// Mitsubishi GX Developer project: PLC_PCO520L2   PLC: Q06UDEH

PROGRAM INPUT
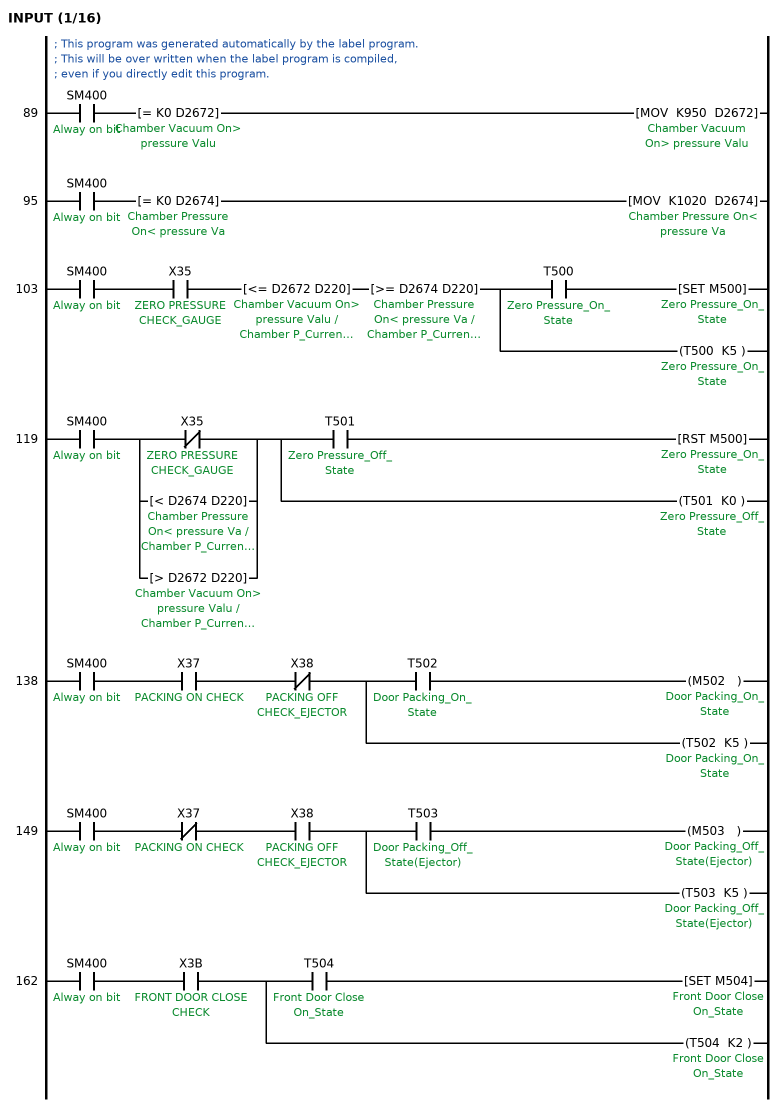
; This program was generated automatically by the label program.
; This will be over written when the label program is compiled,
; even if you directly edit this program.
89    LD      SM400  ; Alway on bit
      AND=    K0 D2672  ; Chamber Vacuum On> pressure Valu
      MOV     K950 D2672
95    LD      SM400  ; Alway on bit
      AND=    K0 D2674  ; Chamber Pressure On< pressure Va
      MOV     K1020 D2674
; 
103   LD      SM400  ; Alway on bit
      AND     X35  ; ZERO PRESSURE CHECK_GAUGE
      AND<=   D2672 D220  ; Chamber Vacuum On> pressure Valu / Chamber P_Current Pressure
      AND>=   D2674 D220  ; Chamber Pressure On< pressure Va / Chamber P_Current Pressure
      MPS
      AND     T500  ; Zero Pressure_On_State
      SET     M500  ; Zero Pressure_On_State
      MPP
      OUT     T500 K5  ; Zero Pressure_On_State
119   LD      SM400  ; Alway on bit
      LDI     X35  ; ZERO PRESSURE CHECK_GAUGE
      OR<     D2674 D220  ; Chamber Pressure On< pressure Va / Chamber P_Current Pressure
      OR>     D2672 D220  ; Chamber Vacuum On> pressure Valu / Chamber P_Current Pressure
      ANB
      MPS
      AND     T501  ; Zero Pressure_Off_State
      RST     M500  ; Zero Pressure_On_State
      MPP
      OUT     T501 K0  ; Zero Pressure_Off_State
; 
138   LD      SM400  ; Alway on bit
      AND     X37  ; PACKING ON CHECK
      ANI     X38  ; PACKING OFF CHECK_EJECTOR
      MPS
      AND     T502  ; Door Packing_On_State
      OUT     M502  ; Door Packing_On_State
      MPP
      OUT     T502 K5  ; Door Packing_On_State
149   LD      SM400  ; Alway on bit
      ANI     X37  ; PACKING ON CHECK
      AND     X38  ; PACKING OFF CHECK_EJECTOR
      MPS
      AND     T503  ; Door Packing_Off_State(Ejector)
      OUT     M503  ; Door Packing_Off_State(Ejector)
      MPP
      OUT     T503 K5  ; Door Packing_Off_State(Ejector)
; 
162   LD      SM400  ; Alway on bit
      AND     X3B  ; FRONT DOOR CLOSE CHECK
      MPS
      AND     T504  ; Front Door Close On_State
      SET     M504  ; Front Door Close On_State
      MPP
      OUT     T504 K2  ; Front Door Close On_State
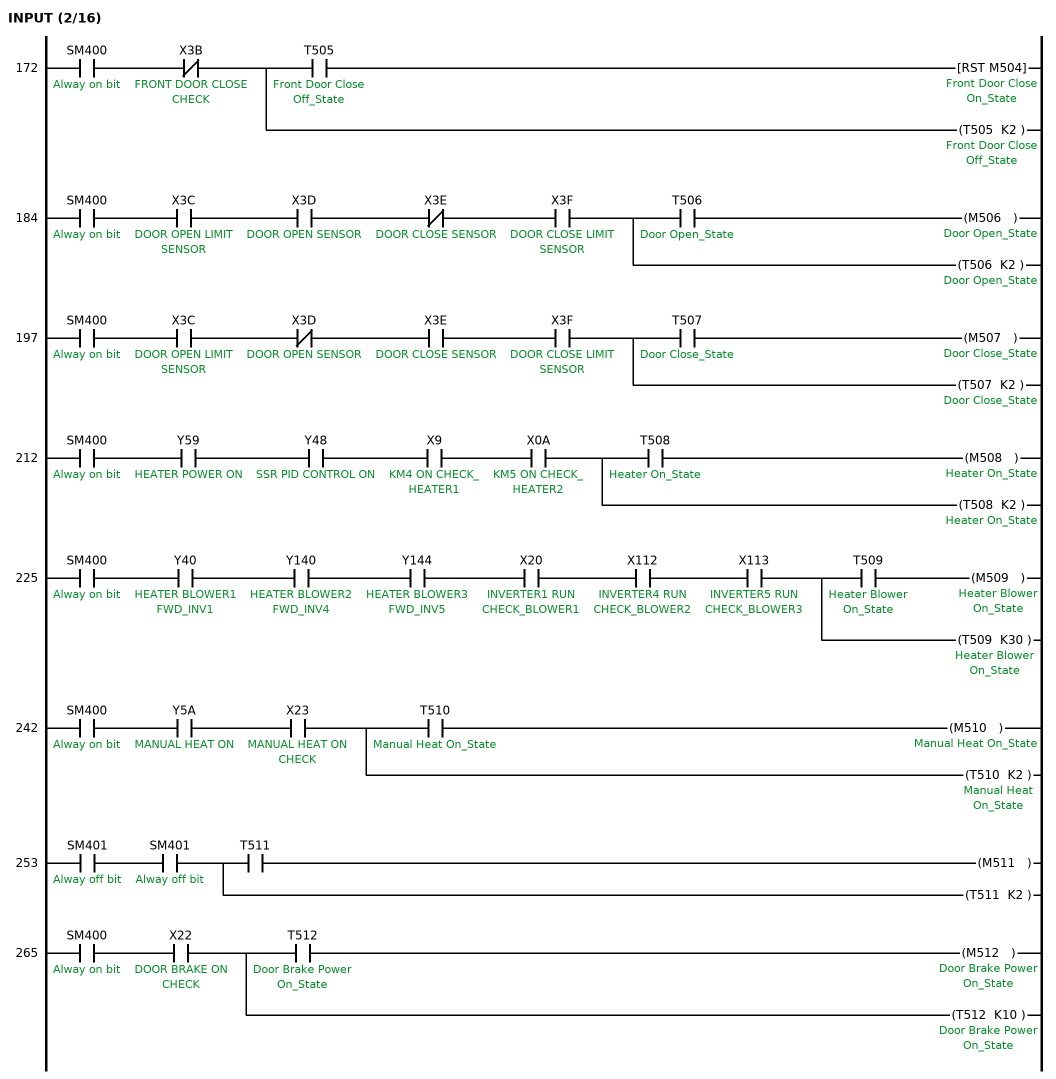
172   LD      SM400  ; Alway on bit
      ANI     X3B  ; FRONT DOOR CLOSE CHECK
      MPS
      AND     T505  ; Front Door Close Off_State
      RST     M504  ; Front Door Close On_State
      MPP
      OUT     T505 K2  ; Front Door Close Off_State
; 
184   LD      SM400  ; Alway on bit
      AND     X3C  ; DOOR OPEN LIMIT SENSOR
      AND     X3D  ; DOOR OPEN SENSOR
      ANI     X3E  ; DOOR CLOSE SENSOR
      AND     X3F  ; DOOR CLOSE LIMIT SENSOR
      MPS
      AND     T506  ; Door Open_State
      OUT     M506  ; Door Open_State
      MPP
      OUT     T506 K2  ; Door Open_State
197   LD      SM400  ; Alway on bit
      AND     X3C  ; DOOR OPEN LIMIT SENSOR
      ANI     X3D  ; DOOR OPEN SENSOR
      AND     X3E  ; DOOR CLOSE SENSOR
      AND     X3F  ; DOOR CLOSE LIMIT SENSOR
      MPS
      AND     T507  ; Door Close_State
      OUT     M507  ; Door Close_State
      MPP
      OUT     T507 K2  ; Door Close_State
; 
212   LD      SM400  ; Alway on bit
      AND     Y59  ; HEATER POWER ON
      AND     Y48  ; SSR PID CONTROL ON
      AND     X9  ; KM4 ON CHECK_HEATER1
      AND     X0A  ; KM5 ON CHECK_HEATER2
      MPS
      AND     T508  ; Heater On_State
      OUT     M508  ; Heater On_State
      MPP
      OUT     T508 K2  ; Heater On_State
225   LD      SM400  ; Alway on bit
      AND     Y40  ; HEATER BLOWER1 FWD_INV1
      AND     Y140  ; HEATER BLOWER2 FWD_INV4
      AND     Y144  ; HEATER BLOWER3 FWD_INV5
      AND     X20  ; INVERTER1 RUN CHECK_BLOWER1
      AND     X112  ; INVERTER4 RUN CHECK_BLOWER2
      AND     X113  ; INVERTER5 RUN CHECK_BLOWER3
      MPS
      AND     T509  ; Heater Blower On_State
      OUT     M509  ; Heater Blower On_State
      MPP
      OUT     T509 K30  ; Heater Blower On_State
; 
242   LD      SM400  ; Alway on bit
      AND     Y5A  ; MANUAL HEAT ON
      AND     X23  ; MANUAL HEAT ON CHECK
      MPS
      AND     T510  ; Manual Heat On_State
      OUT     M510  ; Manual Heat On_State
      MPP
      OUT     T510 K2  ; Manual Heat On_State
253   LD      SM401  ; Alway off bit
      AND     SM401  ; Alway off bit
      MPS
      AND     T511
      OUT     M511
      MPP
      OUT     T511 K2
; 
265   LD      SM400  ; Alway on bit
      AND     X22  ; DOOR BRAKE ON CHECK
      MPS
      AND     T512  ; Door Brake Power On_State
      OUT     M512  ; Door Brake Power On_State
      MPP
      OUT     T512 K10  ; Door Brake Power On_State
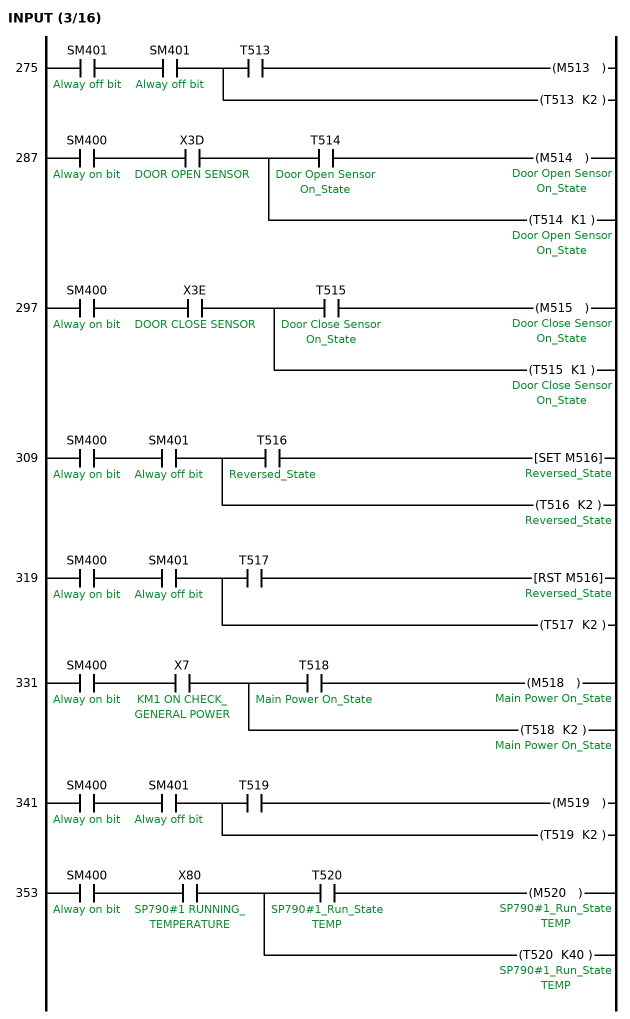
275   LD      SM401  ; Alway off bit
      AND     SM401  ; Alway off bit
      MPS
      AND     T513
      OUT     M513
      MPP
      OUT     T513 K2
; 
287   LD      SM400  ; Alway on bit
      AND     X3D  ; DOOR OPEN SENSOR
      MPS
      AND     T514  ; Door Open Sensor On_State
      OUT     M514  ; Door Open Sensor On_State
      MPP
      OUT     T514 K1  ; Door Open Sensor On_State
297   LD      SM400  ; Alway on bit
      AND     X3E  ; DOOR CLOSE SENSOR
      MPS
      AND     T515  ; Door Close Sensor On_State
      OUT     M515  ; Door Close Sensor On_State
      MPP
      OUT     T515 K1  ; Door Close Sensor On_State
; 
309   LD      SM400  ; Alway on bit
      AND     SM401  ; Alway off bit
      MPS
      AND     T516  ; Reversed_State
      SET     M516  ; Reversed_State
      MPP
      OUT     T516 K2  ; Reversed_State
319   LD      SM400  ; Alway on bit
      AND     SM401  ; Alway off bit
      MPS
      AND     T517
      RST     M516  ; Reversed_State
      MPP
      OUT     T517 K2
; 
331   LD      SM400  ; Alway on bit
      AND     X7  ; KM1 ON CHECK_GENERAL POWER
      MPS
      AND     T518  ; Main Power On_State
      OUT     M518  ; Main Power On_State
      MPP
      OUT     T518 K2  ; Main Power On_State
341   LD      SM400  ; Alway on bit
      AND     SM401  ; Alway off bit
      MPS
      AND     T519
      OUT     M519
      MPP
      OUT     T519 K2
; 
353   LD      SM400  ; Alway on bit
      AND     X80  ; SP790#1 RUNNING_TEMPERATURE
      MPS
      AND     T520  ; SP790#1_Run_State TEMP
      OUT     M520  ; SP790#1_Run_State TEMP
      MPP
      OUT     T520 K40  ; SP790#1_Run_State TEMP
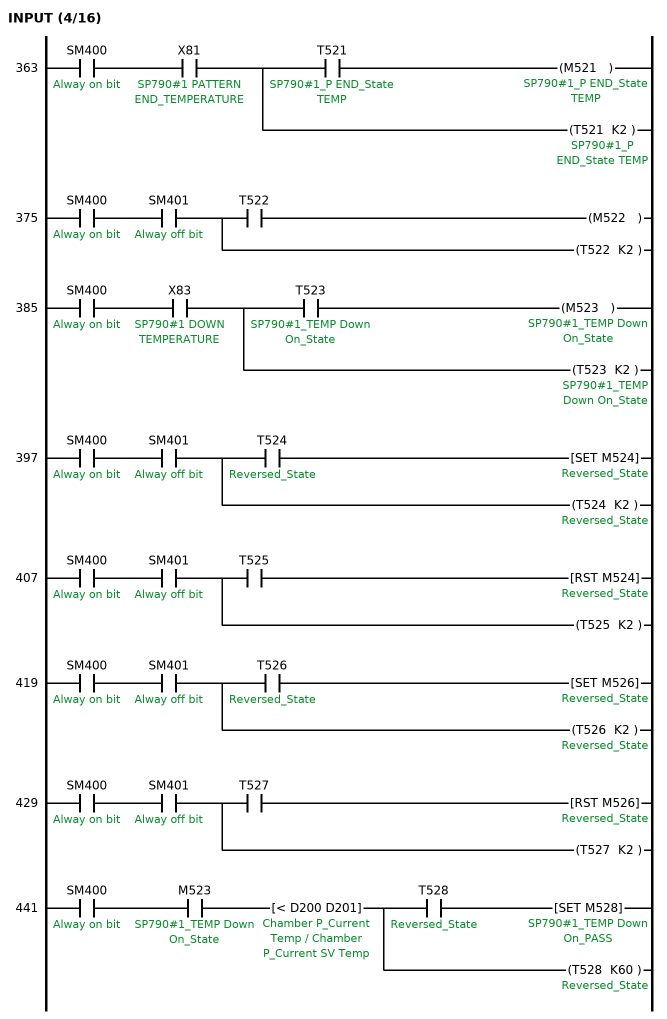
363   LD      SM400  ; Alway on bit
      AND     X81  ; SP790#1 PATTERN END_TEMPERATURE
      MPS
      AND     T521  ; SP790#1_P END_State TEMP
      OUT     M521  ; SP790#1_P END_State TEMP
      MPP
      OUT     T521 K2  ; SP790#1_P END_State TEMP
; 
375   LD      SM400  ; Alway on bit
      AND     SM401  ; Alway off bit
      MPS
      AND     T522
      OUT     M522
      MPP
      OUT     T522 K2
385   LD      SM400  ; Alway on bit
      AND     X83  ; SP790#1 DOWN TEMPERATURE
      MPS
      AND     T523  ; SP790#1_TEMP Down On_State
      OUT     M523  ; SP790#1_TEMP Down On_State
      MPP
      OUT     T523 K2  ; SP790#1_TEMP Down On_State
; 
397   LD      SM400  ; Alway on bit
      AND     SM401  ; Alway off bit
      MPS
      AND     T524  ; Reversed_State
      SET     M524  ; Reversed_State
      MPP
      OUT     T524 K2  ; Reversed_State
407   LD      SM400  ; Alway on bit
      AND     SM401  ; Alway off bit
      MPS
      AND     T525
      RST     M524  ; Reversed_State
      MPP
      OUT     T525 K2
; 
419   LD      SM400  ; Alway on bit
      AND     SM401  ; Alway off bit
      MPS
      AND     T526  ; Reversed_State
      SET     M526  ; Reversed_State
      MPP
      OUT     T526 K2  ; Reversed_State
429   LD      SM400  ; Alway on bit
      AND     SM401  ; Alway off bit
      MPS
      AND     T527
      RST     M526  ; Reversed_State
      MPP
      OUT     T527 K2
; 
441   LD      SM400  ; Alway on bit
      AND     M523  ; SP790#1_TEMP Down On_State
      AND<    D200 D201  ; Chamber P_Current Temp / Chamber P_Current SV Temp
      MPS
      AND     T528  ; Reversed_State
      SET     M528  ; SP790#1_TEMP Down On_PASS
      MPP
      OUT     T528 K60  ; Reversed_State
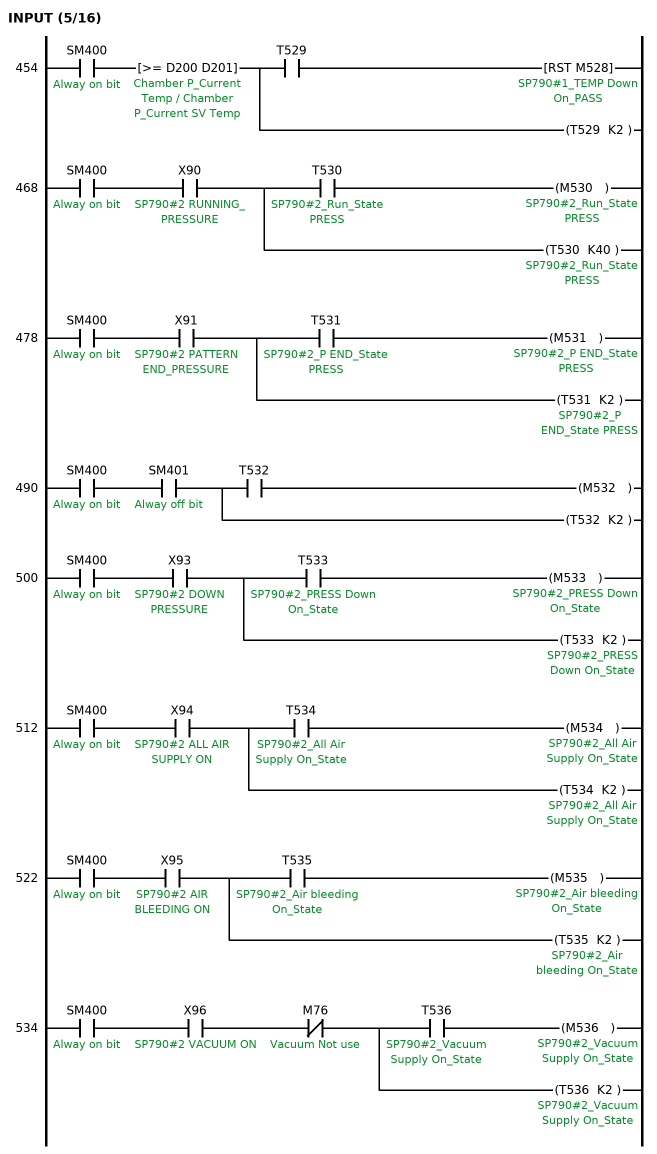
454   LD      SM400  ; Alway on bit
      AND>=   D200 D201  ; Chamber P_Current Temp / Chamber P_Current SV Temp
      MPS
      AND     T529
      RST     M528  ; SP790#1_TEMP Down On_PASS
      MPP
      OUT     T529 K2
; 
468   LD      SM400  ; Alway on bit
      AND     X90  ; SP790#2 RUNNING_PRESSURE
      MPS
      AND     T530  ; SP790#2_Run_State PRESS
      OUT     M530  ; SP790#2_Run_State PRESS
      MPP
      OUT     T530 K40  ; SP790#2_Run_State PRESS
478   LD      SM400  ; Alway on bit
      AND     X91  ; SP790#2 PATTERN END_PRESSURE
      MPS
      AND     T531  ; SP790#2_P END_State PRESS
      OUT     M531  ; SP790#2_P END_State PRESS
      MPP
      OUT     T531 K2  ; SP790#2_P END_State PRESS
; 
490   LD      SM400  ; Alway on bit
      AND     SM401  ; Alway off bit
      MPS
      AND     T532
      OUT     M532
      MPP
      OUT     T532 K2
500   LD      SM400  ; Alway on bit
      AND     X93  ; SP790#2 DOWN PRESSURE
      MPS
      AND     T533  ; SP790#2_PRESS Down On_State
      OUT     M533  ; SP790#2_PRESS Down On_State
      MPP
      OUT     T533 K2  ; SP790#2_PRESS Down On_State
; 
512   LD      SM400  ; Alway on bit
      AND     X94  ; SP790#2 ALL AIR SUPPLY ON
      MPS
      AND     T534  ; SP790#2_All Air Supply On_State
      OUT     M534  ; SP790#2_All Air Supply On_State
      MPP
      OUT     T534 K2  ; SP790#2_All Air Supply On_State
522   LD      SM400  ; Alway on bit
      AND     X95  ; SP790#2 AIR BLEEDING ON
      MPS
      AND     T535  ; SP790#2_Air bleeding On_State
      OUT     M535  ; SP790#2_Air bleeding On_State
      MPP
      OUT     T535 K2  ; SP790#2_Air bleeding On_State
; 
534   LD      SM400  ; Alway on bit
      AND     X96  ; SP790#2 VACUUM ON
      ANI     M76  ; Vacuum Not use
      MPS
      AND     T536  ; SP790#2_Vacuum Supply On_State
      OUT     M536  ; SP790#2_Vacuum Supply On_State
      MPP
      OUT     T536 K2  ; SP790#2_Vacuum Supply On_State
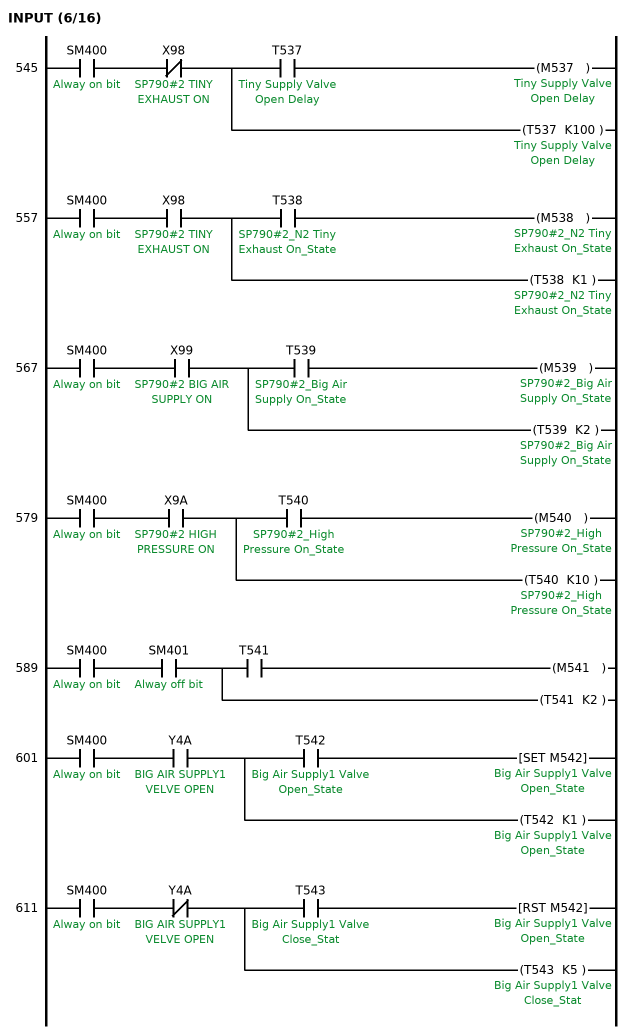
545   LD      SM400  ; Alway on bit
      ANI     X98  ; SP790#2 TINY EXHAUST ON
      MPS
      AND     T537  ; Tiny Supply Valve Open Delay
      OUT     M537  ; Tiny Supply Valve Open Delay
      MPP
      OUT     T537 K100  ; Tiny Supply Valve Open Delay
; 
557   LD      SM400  ; Alway on bit
      AND     X98  ; SP790#2 TINY EXHAUST ON
      MPS
      AND     T538  ; SP790#2_N2 Tiny Exhaust On_State
      OUT     M538  ; SP790#2_N2 Tiny Exhaust On_State
      MPP
      OUT     T538 K1  ; SP790#2_N2 Tiny Exhaust On_State
567   LD      SM400  ; Alway on bit
      AND     X99  ; SP790#2 BIG AIR SUPPLY ON
      MPS
      AND     T539  ; SP790#2_Big Air Supply On_State
      OUT     M539  ; SP790#2_Big Air Supply On_State
      MPP
      OUT     T539 K2  ; SP790#2_Big Air Supply On_State
; 
579   LD      SM400  ; Alway on bit
      AND     X9A  ; SP790#2 HIGH PRESSURE ON
      MPS
      AND     T540  ; SP790#2_High Pressure On_State
      OUT     M540  ; SP790#2_High Pressure On_State
      MPP
      OUT     T540 K10  ; SP790#2_High Pressure On_State
589   LD      SM400  ; Alway on bit
      AND     SM401  ; Alway off bit
      MPS
      AND     T541
      OUT     M541
      MPP
      OUT     T541 K2
; 
601   LD      SM400  ; Alway on bit
      AND     Y4A  ; BIG AIR SUPPLY1 VELVE OPEN
      MPS
      AND     T542  ; Big Air Supply1 Valve Open_State
      SET     M542  ; Big Air Supply1 Valve Open_State
      MPP
      OUT     T542 K1  ; Big Air Supply1 Valve Open_State
611   LD      SM400  ; Alway on bit
      ANI     Y4A  ; BIG AIR SUPPLY1 VELVE OPEN
      MPS
      AND     T543  ; Big Air Supply1 Valve Close_Stat
      RST     M542  ; Big Air Supply1 Valve Open_State
      MPP
      OUT     T543 K5  ; Big Air Supply1 Valve Close_Stat
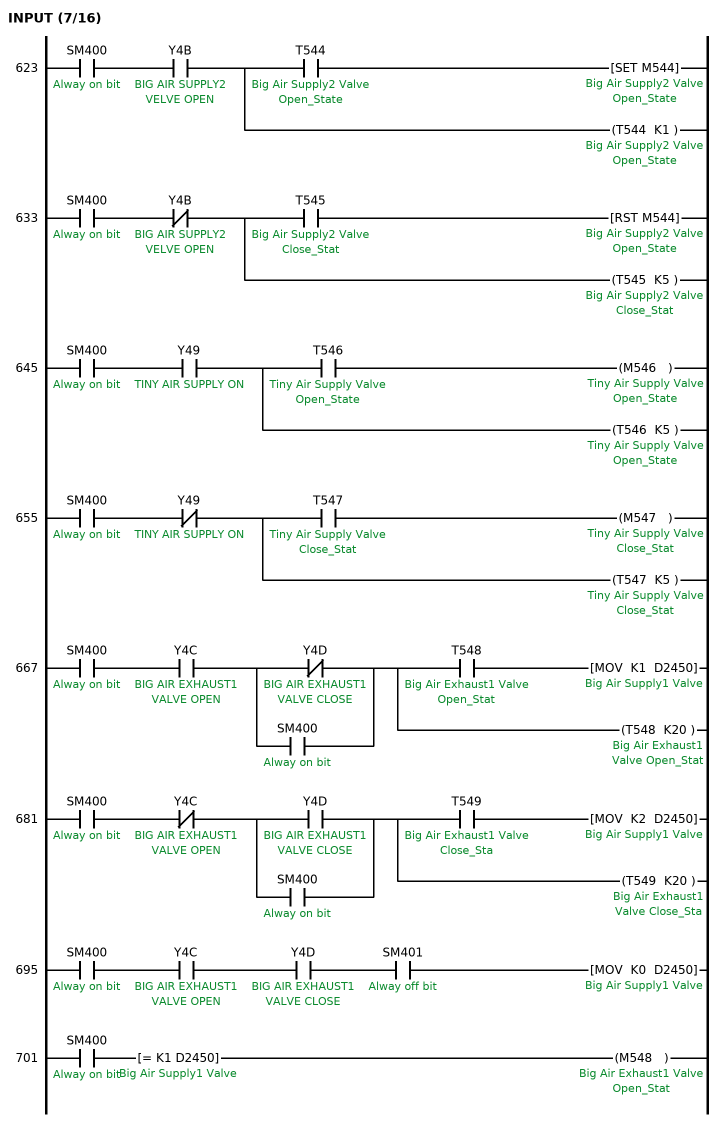
; 
623   LD      SM400  ; Alway on bit
      AND     Y4B  ; BIG AIR SUPPLY2 VELVE OPEN
      MPS
      AND     T544  ; Big Air Supply2 Valve Open_State
      SET     M544  ; Big Air Supply2 Valve Open_State
      MPP
      OUT     T544 K1  ; Big Air Supply2 Valve Open_State
633   LD      SM400  ; Alway on bit
      ANI     Y4B  ; BIG AIR SUPPLY2 VELVE OPEN
      MPS
      AND     T545  ; Big Air Supply2 Valve Close_Stat
      RST     M544  ; Big Air Supply2 Valve Open_State
      MPP
      OUT     T545 K5  ; Big Air Supply2 Valve Close_Stat
; 
645   LD      SM400  ; Alway on bit
      AND     Y49  ; TINY AIR SUPPLY ON
      MPS
      AND     T546  ; Tiny Air Supply Valve Open_State
      OUT     M546  ; Tiny Air Supply Valve Open_State
      MPP
      OUT     T546 K5  ; Tiny Air Supply Valve Open_State
655   LD      SM400  ; Alway on bit
      ANI     Y49  ; TINY AIR SUPPLY ON
      MPS
      AND     T547  ; Tiny Air Supply Valve Close_Stat
      OUT     M547  ; Tiny Air Supply Valve Close_Stat
      MPP
      OUT     T547 K5  ; Tiny Air Supply Valve Close_Stat
; 
667   LD      SM400  ; Alway on bit
      AND     Y4C  ; BIG AIR EXHAUST1 VALVE OPEN
      LDI     Y4D  ; BIG AIR EXHAUST1 VALVE CLOSE
      OR      SM400  ; Alway on bit
      ANB
      MPS
      AND     T548  ; Big Air Exhaust1 Valve Open_Stat
      MOV     K1 D2450  ; Big Air Supply1 Valve
      MPP
      OUT     T548 K20  ; Big Air Exhaust1 Valve Open_Stat
681   LD      SM400  ; Alway on bit
      ANI     Y4C  ; BIG AIR EXHAUST1 VALVE OPEN
      LD      Y4D  ; BIG AIR EXHAUST1 VALVE CLOSE
      OR      SM400  ; Alway on bit
      ANB
      MPS
      AND     T549  ; Big Air Exhaust1 Valve Close_Sta
      MOV     K2 D2450
      MPP
      OUT     T549 K20  ; Big Air Exhaust1 Valve Close_Sta
695   LD      SM400  ; Alway on bit
      AND     Y4C  ; BIG AIR EXHAUST1 VALVE OPEN
      AND     Y4D  ; BIG AIR EXHAUST1 VALVE CLOSE
      AND     SM401  ; Alway off bit
      MOV     K0 D2450
701   LD      SM400  ; Alway on bit
      AND=    K1 D2450  ; Big Air Supply1 Valve
      OUT     M548  ; Big Air Exhaust1 Valve Open_Stat
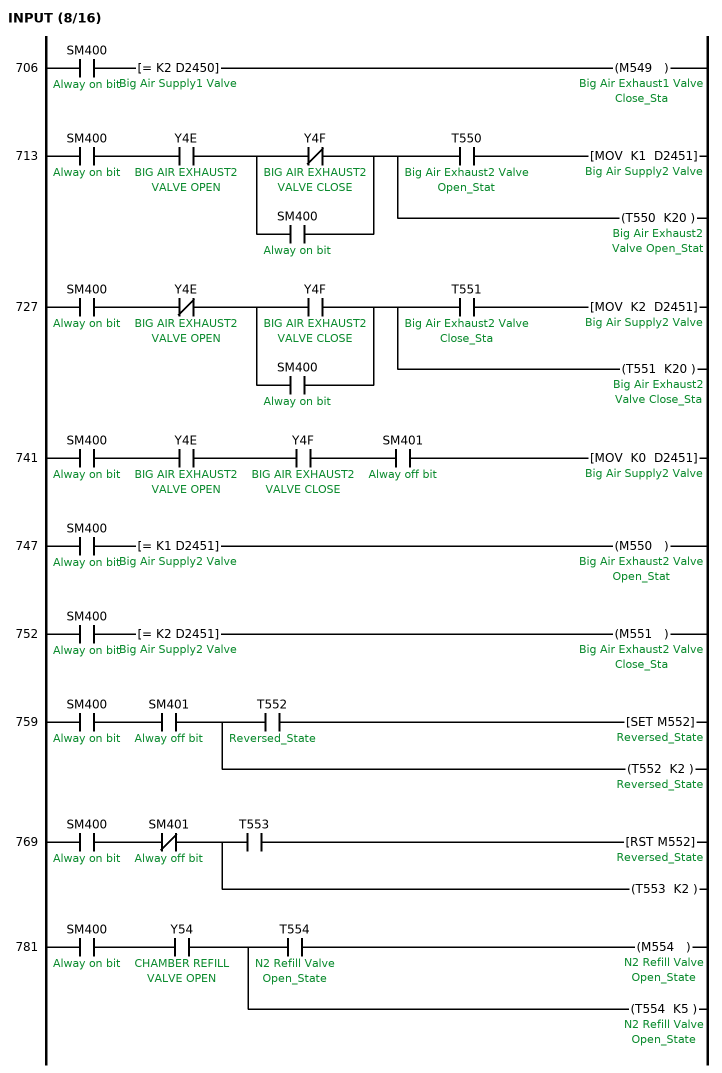
706   LD      SM400  ; Alway on bit
      AND=    K2 D2450  ; Big Air Supply1 Valve
      OUT     M549  ; Big Air Exhaust1 Valve Close_Sta
; 
713   LD      SM400  ; Alway on bit
      AND     Y4E  ; BIG AIR EXHAUST2 VALVE OPEN
      LDI     Y4F  ; BIG AIR EXHAUST2 VALVE CLOSE
      OR      SM400  ; Alway on bit
      ANB
      MPS
      AND     T550  ; Big Air Exhaust2 Valve Open_Stat
      MOV     K1 D2451  ; Big Air Supply2 Valve
      MPP
      OUT     T550 K20  ; Big Air Exhaust2 Valve Open_Stat
727   LD      SM400  ; Alway on bit
      ANI     Y4E  ; BIG AIR EXHAUST2 VALVE OPEN
      LD      Y4F  ; BIG AIR EXHAUST2 VALVE CLOSE
      OR      SM400  ; Alway on bit
      ANB
      MPS
      AND     T551  ; Big Air Exhaust2 Valve Close_Sta
      MOV     K2 D2451
      MPP
      OUT     T551 K20  ; Big Air Exhaust2 Valve Close_Sta
741   LD      SM400  ; Alway on bit
      AND     Y4E  ; BIG AIR EXHAUST2 VALVE OPEN
      AND     Y4F  ; BIG AIR EXHAUST2 VALVE CLOSE
      AND     SM401  ; Alway off bit
      MOV     K0 D2451
747   LD      SM400  ; Alway on bit
      AND=    K1 D2451  ; Big Air Supply2 Valve
      OUT     M550  ; Big Air Exhaust2 Valve Open_Stat
752   LD      SM400  ; Alway on bit
      AND=    K2 D2451  ; Big Air Supply2 Valve
      OUT     M551  ; Big Air Exhaust2 Valve Close_Sta
; 
759   LD      SM400  ; Alway on bit
      AND     SM401  ; Alway off bit
      MPS
      AND     T552  ; Reversed_State
      SET     M552  ; Reversed_State
      MPP
      OUT     T552 K2  ; Reversed_State
769   LD      SM400  ; Alway on bit
      ANI     SM401  ; Alway off bit
      MPS
      AND     T553
      RST     M552  ; Reversed_State
      MPP
      OUT     T553 K2
; 
781   LD      SM400  ; Alway on bit
      AND     Y54  ; CHAMBER REFILL VALVE OPEN
      MPS
      AND     T554  ; N2 Refill Valve Open_State
      OUT     M554  ; N2 Refill Valve Open_State
      MPP
      OUT     T554 K5  ; N2 Refill Valve Open_State
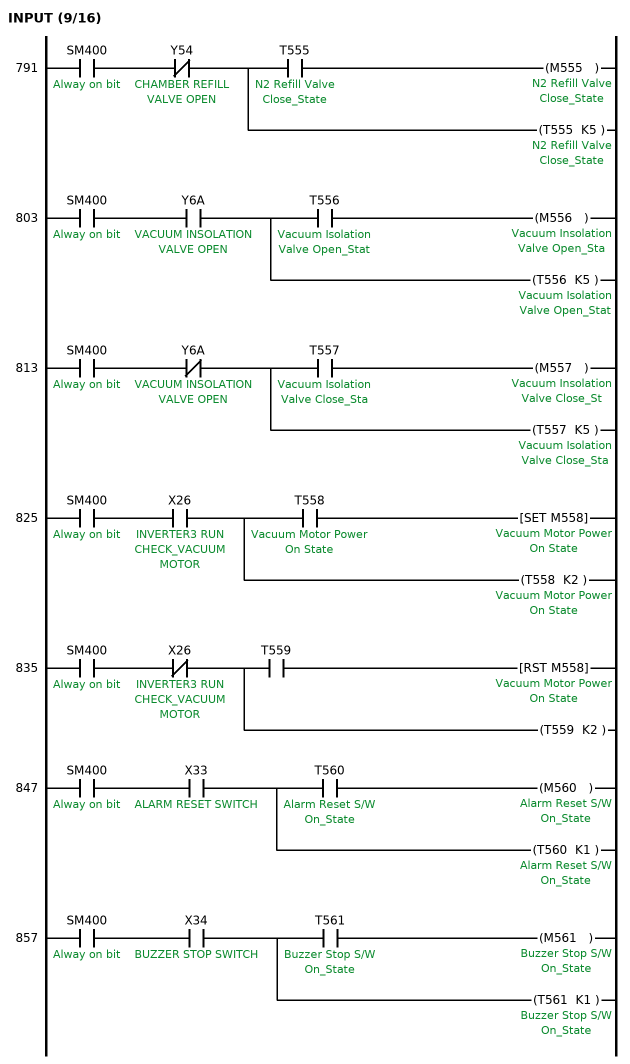
791   LD      SM400  ; Alway on bit
      ANI     Y54  ; CHAMBER REFILL VALVE OPEN
      MPS
      AND     T555  ; N2 Refill Valve Close_State
      OUT     M555  ; N2 Refill Valve Close_State
      MPP
      OUT     T555 K5  ; N2 Refill Valve Close_State
; 
803   LD      SM400  ; Alway on bit
      AND     Y6A  ; VACUUM INSOLATION VALVE OPEN
      MPS
      AND     T556  ; Vacuum Isolation Valve Open_Stat
      OUT     M556  ; Vacuum Insolation Valve Open_Sta
      MPP
      OUT     T556 K5  ; Vacuum Isolation Valve Open_Stat
813   LD      SM400  ; Alway on bit
      ANI     Y6A  ; VACUUM INSOLATION VALVE OPEN
      MPS
      AND     T557  ; Vacuum Isolation Valve Close_Sta
      OUT     M557  ; Vacuum Insolation Valve Close_St
      MPP
      OUT     T557 K5  ; Vacuum Isolation Valve Close_Sta
; 
825   LD      SM400  ; Alway on bit
      AND     X26  ; INVERTER3 RUN CHECK_VACUUM MOTOR
      MPS
      AND     T558  ; Vacuum Motor Power On State
      SET     M558  ; Vacuum Motor Power On State
      MPP
      OUT     T558 K2  ; Vacuum Motor Power On State
835   LD      SM400  ; Alway on bit
      ANI     X26  ; INVERTER3 RUN CHECK_VACUUM MOTOR
      MPS
      AND     T559
      RST     M558  ; Vacuum Motor Power On State
      MPP
      OUT     T559 K2
; 
847   LD      SM400  ; Alway on bit
      AND     X33  ; ALARM RESET SWITCH
      MPS
      AND     T560  ; Alarm Reset S/W On_State
      OUT     M560  ; Alarm Reset S/W On_State
      MPP
      OUT     T560 K1  ; Alarm Reset S/W On_State
857   LD      SM400  ; Alway on bit
      AND     X34  ; BUZZER STOP SWITCH
      MPS
      AND     T561  ; Buzzer Stop S/W On_State
      OUT     M561  ; Buzzer Stop S/W On_State
      MPP
      OUT     T561 K1  ; Buzzer Stop S/W On_State
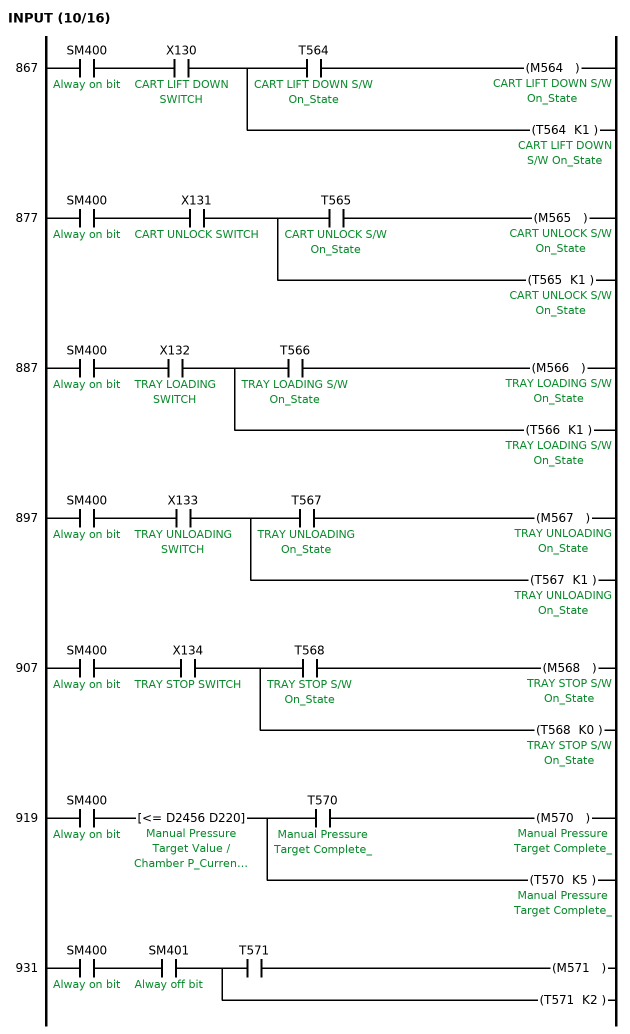
867   LD      SM400  ; Alway on bit
      AND     X130  ; CART LIFT DOWN SWITCH
      MPS
      AND     T564  ; CART LIFT DOWN S/W On_State
      OUT     M564  ; CART LIFT DOWN S/W On_State
      MPP
      OUT     T564 K1  ; CART LIFT DOWN S/W On_State
877   LD      SM400  ; Alway on bit
      AND     X131  ; CART UNLOCK SWITCH
      MPS
      AND     T565  ; CART UNLOCK S/W On_State
      OUT     M565  ; CART UNLOCK S/W On_State
      MPP
      OUT     T565 K1  ; CART UNLOCK S/W On_State
887   LD      SM400  ; Alway on bit
      AND     X132  ; TRAY LOADING SWITCH
      MPS
      AND     T566  ; TRAY LOADING S/W On_State
      OUT     M566  ; TRAY LOADING S/W On_State
      MPP
      OUT     T566 K1  ; TRAY LOADING S/W On_State
897   LD      SM400  ; Alway on bit
      AND     X133  ; TRAY UNLOADING SWITCH
      MPS
      AND     T567  ; TRAY UNLOADING On_State
      OUT     M567  ; TRAY UNLOADING On_State
      MPP
      OUT     T567 K1  ; TRAY UNLOADING On_State
907   LD      SM400  ; Alway on bit
      AND     X134  ; TRAY STOP SWITCH
      MPS
      AND     T568  ; TRAY STOP S/W On_State
      OUT     M568  ; TRAY STOP S/W On_State
      MPP
      OUT     T568 K0  ; TRAY STOP S/W On_State
; 
919   LD      SM400  ; Alway on bit
      AND<=   D2456 D220  ; Manual Pressure Target Value / Chamber P_Current Pressure
      MPS
      AND     T570  ; Manual Pressure Target Complete_
      OUT     M570  ; Manual Pressure Target Complete_
      MPP
      OUT     T570 K5  ; Manual Pressure Target Complete_
931   LD      SM400  ; Alway on bit
      AND     SM401  ; Alway off bit
      MPS
      AND     T571
      OUT     M571
      MPP
      OUT     T571 K2
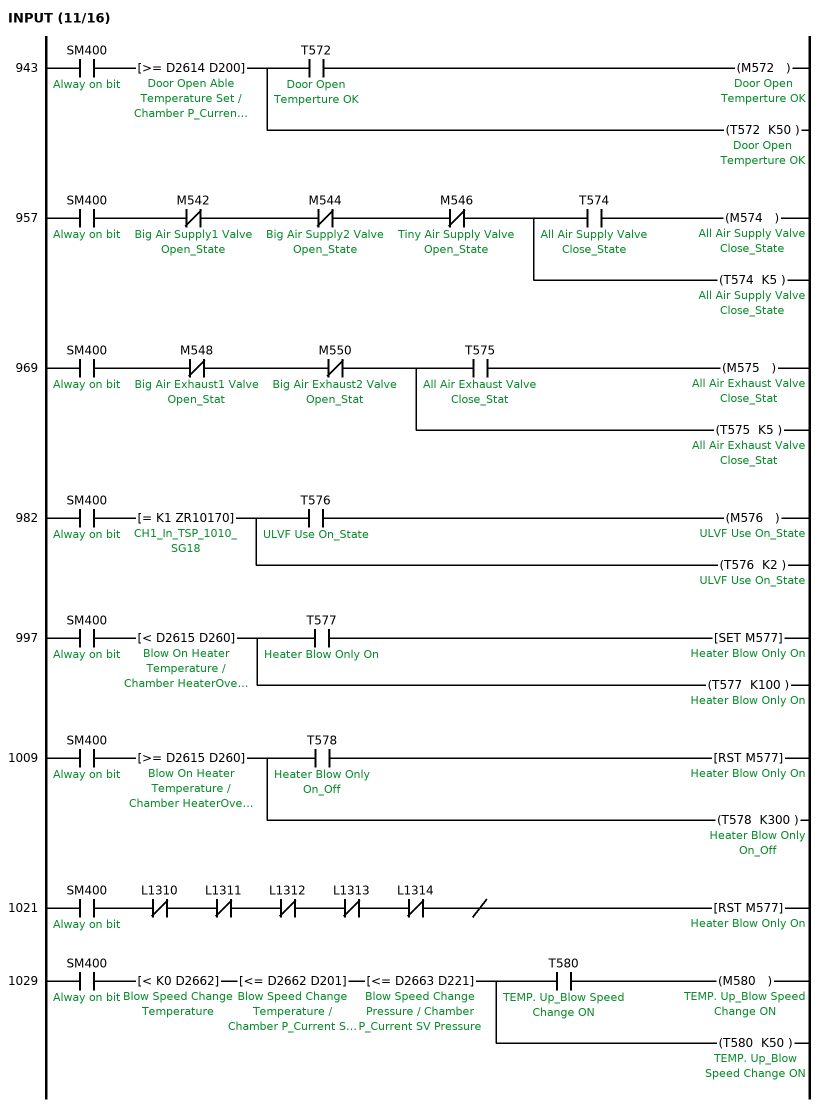
; 
943   LD      SM400  ; Alway on bit
      AND>=   D2614 D200  ; Door Open Able Temperature Set / Chamber P_Current Temp
      MPS
      AND     T572  ; Door Open Temperture OK
      OUT     M572  ; Door Open Temperture OK
      MPP
      OUT     T572 K50  ; Door Open Temperture OK
; 
957   LD      SM400  ; Alway on bit
      ANI     M542  ; Big Air Supply1 Valve Open_State
      ANI     M544  ; Big Air Supply2 Valve Open_State
      ANI     M546  ; Tiny Air Supply Valve Open_State
      MPS
      AND     T574  ; All Air Supply Valve Close_State
      OUT     M574  ; All Air Supply Valve Close_State
      MPP
      OUT     T574 K5  ; All Air Supply Valve Close_State
969   LD      SM400  ; Alway on bit
      ANI     M548  ; Big Air Exhaust1 Valve Open_Stat
      ANI     M550  ; Big Air Exhaust2 Valve Open_Stat
      MPS
      AND     T575  ; All Air Exhaust Valve Close_Stat
      OUT     M575  ; All Air Exhaust Valve Close_Stat
      MPP
      OUT     T575 K5  ; All Air Exhaust Valve Close_Stat
; 
982   LD      SM400  ; Alway on bit
      AND=    K1 ZR10170  ; CH1_In_TSP_1010_SG18
      MPS
      AND     T576  ; ULVF Use On_State
      OUT     M576  ; ULVF Use On_State
      MPP
      OUT     T576 K2  ; ULVF Use On_State
; 
997   LD      SM400  ; Alway on bit
      AND<    D2615 D260  ; Blow On Heater Temperature / Chamber HeaterOver Current Temp
      MPS
      AND     T577  ; Heater Blow Only On
      SET     M577  ; Heater Blow Only On
      MPP
      OUT     T577 K100  ; Heater Blow Only On
1009  LD      SM400  ; Alway on bit
      AND>=   D2615 D260  ; Blow On Heater Temperature / Chamber HeaterOver Current Temp
      MPS
      AND     T578  ; Heater Blow Only On_Off
      RST     M577  ; Heater Blow Only On
      MPP
      OUT     T578 K300  ; Heater Blow Only On_Off
1021  LD      SM400  ; Alway on bit
      ANI     L1310
      ANI     L1311
      ANI     L1312
      ANI     L1313
      ANI     L1314
      INV
      RST     M577  ; Heater Blow Only On
1029  LD      SM400  ; Alway on bit
      AND<    K0 D2662  ; Blow Speed Change Temperature
      AND<=   D2662 D201  ; Blow Speed Change Temperature / Chamber P_Current SV Temp
      AND<=   D2663 D221  ; Blow Speed Change Pressure / Chamber P_Current SV Pressure
      MPS
      AND     T580  ; TEMP. Up_Blow Speed Change ON
      OUT     M580  ; TEMP. Up_Blow Speed Change ON
      MPP
      OUT     T580 K50  ; TEMP. Up_Blow Speed Change ON
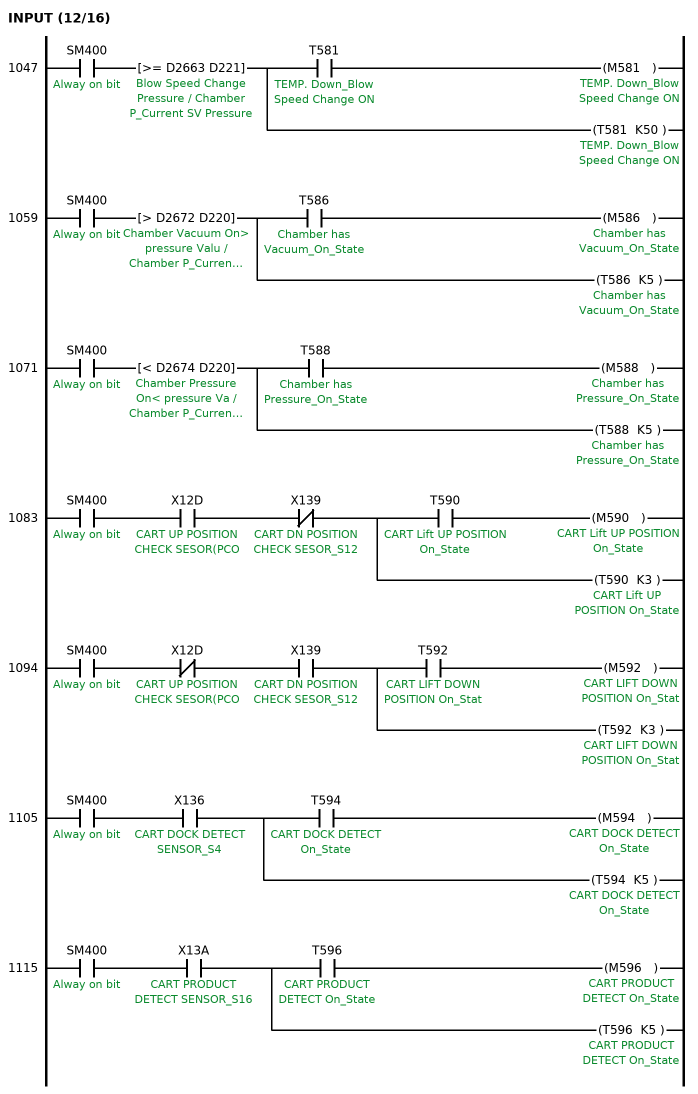
1047  LD      SM400  ; Alway on bit
      AND>=   D2663 D221  ; Blow Speed Change Pressure / Chamber P_Current SV Pressure
      MPS
      AND     T581  ; TEMP. Down_Blow Speed Change ON
      OUT     M581  ; TEMP. Down_Blow Speed Change ON
      MPP
      OUT     T581 K50  ; TEMP. Down_Blow Speed Change ON
1059  LD      SM400  ; Alway on bit
      AND>    D2672 D220  ; Chamber Vacuum On> pressure Valu / Chamber P_Current Pressure
      MPS
      AND     T586  ; Chamber has Vacuum_On_State
      OUT     M586  ; Chamber has Vacuum_On_State
      MPP
      OUT     T586 K5  ; Chamber has Vacuum_On_State
1071  LD      SM400  ; Alway on bit
      AND<    D2674 D220  ; Chamber Pressure On< pressure Va / Chamber P_Current Pressure
      MPS
      AND     T588  ; Chamber has Pressure_On_State
      OUT     M588  ; Chamber has Pressure_On_State
      MPP
      OUT     T588 K5  ; Chamber has Pressure_On_State
1083  LD      SM400  ; Alway on bit
      AND     X12D  ; CART UP POSITION CHECK SESOR(PCO
      ANI     X139  ; CART DN POSITION CHECK SESOR_S12
      MPS
      AND     T590  ; CART Lift UP POSITION On_State
      OUT     M590  ; CART Lift UP POSITION On_State
      MPP
      OUT     T590 K3  ; CART Lift UP POSITION On_State
1094  LD      SM400  ; Alway on bit
      ANI     X12D  ; CART UP POSITION CHECK SESOR(PCO
      AND     X139  ; CART DN POSITION CHECK SESOR_S12
      MPS
      AND     T592  ; CART LIFT DOWN  POSITION On_Stat
      OUT     M592  ; CART LIFT DOWN  POSITION On_Stat
      MPP
      OUT     T592 K3  ; CART LIFT DOWN  POSITION On_Stat
1105  LD      SM400  ; Alway on bit
      AND     X136  ; CART DOCK DETECT SENSOR_S4
      MPS
      AND     T594  ; CART DOCK DETECT On_State
      OUT     M594  ; CART DOCK DETECT On_State
      MPP
      OUT     T594 K5  ; CART DOCK DETECT On_State
1115  LD      SM400  ; Alway on bit
      AND     X13A  ; CART PRODUCT DETECT SENSOR_S16
      MPS
      AND     T596  ; CART PRODUCT DETECT On_State
      OUT     M596  ; CART PRODUCT DETECT On_State
      MPP
      OUT     T596 K5  ; CART PRODUCT DETECT On_State
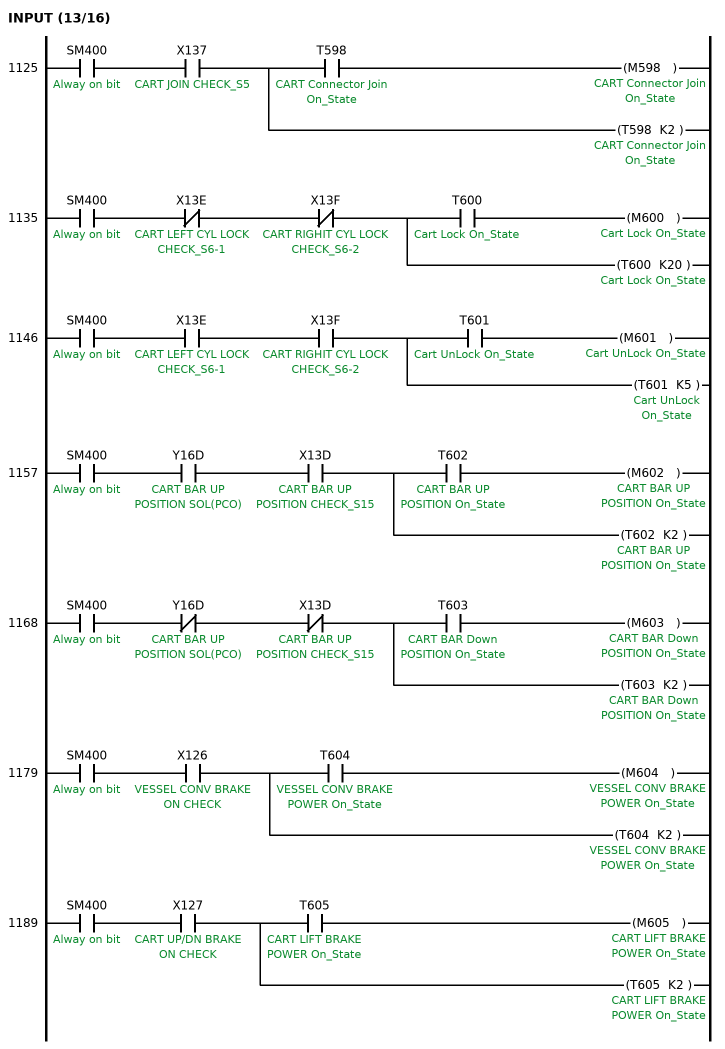
1125  LD      SM400  ; Alway on bit
      AND     X137  ; CART JOIN CHECK_S5
      MPS
      AND     T598  ; CART Connector Join On_State
      OUT     M598  ; CART Connector Join On_State
      MPP
      OUT     T598 K2  ; CART Connector Join On_State
1135  LD      SM400  ; Alway on bit
      ANI     X13E  ; CART LEFT CYL LOCK CHECK_S6-1
      ANI     X13F  ; CART RIGHIT CYL LOCK CHECK_S6-2
      MPS
      AND     T600  ; Cart Lock On_State
      OUT     M600  ; Cart Lock On_State
      MPP
      OUT     T600 K20  ; Cart Lock On_State
1146  LD      SM400  ; Alway on bit
      AND     X13E  ; CART LEFT CYL LOCK CHECK_S6-1
      AND     X13F  ; CART RIGHIT CYL LOCK CHECK_S6-2
      MPS
      AND     T601  ; Cart UnLock On_State
      OUT     M601  ; Cart UnLock On_State
      MPP
      OUT     T601 K5  ; Cart UnLock On_State
1157  LD      SM400  ; Alway on bit
      AND     Y16D  ; CART BAR UP POSITION SOL(PCO)
      AND     X13D  ; CART BAR UP POSITION CHECK_S15
      MPS
      AND     T602  ; CART BAR UP POSITION On_State
      OUT     M602  ; CART BAR UP POSITION On_State
      MPP
      OUT     T602 K2  ; CART BAR UP POSITION On_State
1168  LD      SM400  ; Alway on bit
      ANI     Y16D  ; CART BAR UP POSITION SOL(PCO)
      ANI     X13D  ; CART BAR UP POSITION CHECK_S15
      MPS
      AND     T603  ; CART BAR Down POSITION On_State
      OUT     M603  ; CART BAR Down POSITION On_State
      MPP
      OUT     T603 K2  ; CART BAR Down POSITION On_State
1179  LD      SM400  ; Alway on bit
      AND     X126  ; VESSEL CONV BRAKE ON CHECK
      MPS
      AND     T604  ; VESSEL CONV BRAKE POWER On_State
      OUT     M604  ; VESSEL CONV BRAKE POWER On_State
      MPP
      OUT     T604 K2  ; VESSEL CONV BRAKE POWER On_State
1189  LD      SM400  ; Alway on bit
      AND     X127  ; CART UP/DN BRAKE ON CHECK
      MPS
      AND     T605  ; CART LIFT BRAKE POWER On_State
      OUT     M605  ; CART LIFT BRAKE POWER On_State
      MPP
      OUT     T605 K2  ; CART LIFT BRAKE POWER On_State
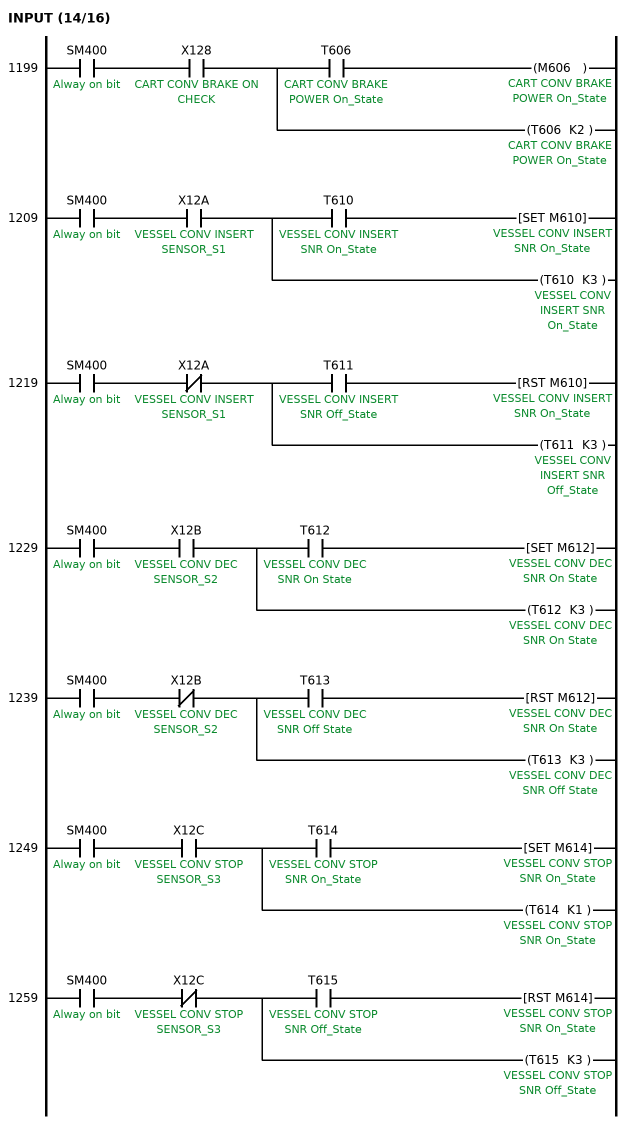
1199  LD      SM400  ; Alway on bit
      AND     X128  ; CART CONV BRAKE ON CHECK
      MPS
      AND     T606  ; CART CONV BRAKE POWER On_State
      OUT     M606  ; CART CONV BRAKE POWER On_State
      MPP
      OUT     T606 K2  ; CART CONV BRAKE POWER On_State
1209  LD      SM400  ; Alway on bit
      AND     X12A  ; VESSEL CONV INSERT SENSOR_S1
      MPS
      AND     T610  ; VESSEL CONV INSERT SNR On_State
      SET     M610  ; VESSEL CONV INSERT SNR On_State
      MPP
      OUT     T610 K3  ; VESSEL CONV INSERT SNR On_State
1219  LD      SM400  ; Alway on bit
      ANI     X12A  ; VESSEL CONV INSERT SENSOR_S1
      MPS
      AND     T611  ; VESSEL CONV INSERT SNR Off_State
      RST     M610  ; VESSEL CONV INSERT SNR On_State
      MPP
      OUT     T611 K3  ; VESSEL CONV INSERT SNR Off_State
1229  LD      SM400  ; Alway on bit
      AND     X12B  ; VESSEL CONV DEC SENSOR_S2
      MPS
      AND     T612  ; VESSEL CONV DEC SNR On State
      SET     M612  ; VESSEL CONV DEC SNR On State
      MPP
      OUT     T612 K3  ; VESSEL CONV DEC SNR On State
1239  LD      SM400  ; Alway on bit
      ANI     X12B  ; VESSEL CONV DEC SENSOR_S2
      MPS
      AND     T613  ; VESSEL CONV DEC SNR Off State
      RST     M612  ; VESSEL CONV DEC SNR On State
      MPP
      OUT     T613 K3  ; VESSEL CONV DEC SNR Off State
1249  LD      SM400  ; Alway on bit
      AND     X12C  ; VESSEL CONV STOP SENSOR_S3
      MPS
      AND     T614  ; VESSEL CONV STOP SNR On_State
      SET     M614  ; VESSEL CONV STOP SNR On_State
      MPP
      OUT     T614 K1  ; VESSEL CONV STOP SNR On_State
1259  LD      SM400  ; Alway on bit
      ANI     X12C  ; VESSEL CONV STOP SENSOR_S3
      MPS
      AND     T615  ; VESSEL CONV STOP SNR Off_State
      RST     M614  ; VESSEL CONV STOP SNR On_State
      MPP
      OUT     T615 K3  ; VESSEL CONV STOP SNR Off_State
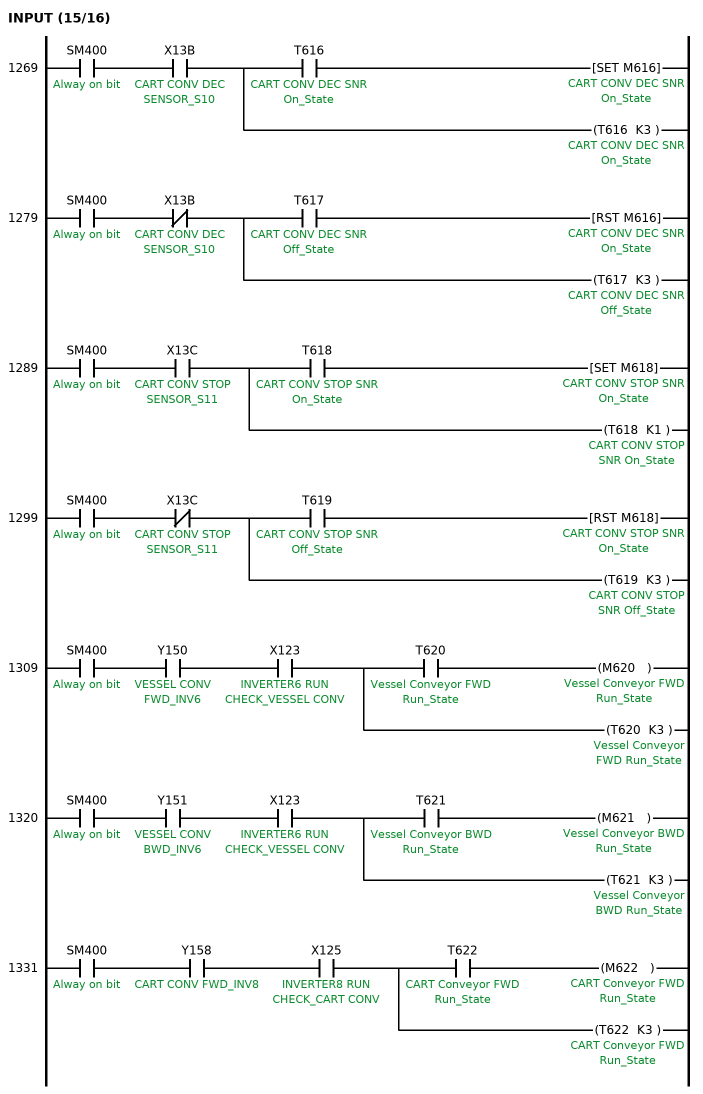
1269  LD      SM400  ; Alway on bit
      AND     X13B  ; CART CONV DEC SENSOR_S10
      MPS
      AND     T616  ; CART CONV DEC SNR On_State
      SET     M616  ; CART CONV DEC SNR On_State
      MPP
      OUT     T616 K3  ; CART CONV DEC SNR On_State
1279  LD      SM400  ; Alway on bit
      ANI     X13B  ; CART CONV DEC SENSOR_S10
      MPS
      AND     T617  ; CART CONV DEC SNR Off_State
      RST     M616  ; CART CONV DEC SNR On_State
      MPP
      OUT     T617 K3  ; CART CONV DEC SNR Off_State
1289  LD      SM400  ; Alway on bit
      AND     X13C  ; CART CONV STOP SENSOR_S11
      MPS
      AND     T618  ; CART CONV STOP SNR On_State
      SET     M618  ; CART CONV STOP SNR On_State
      MPP
      OUT     T618 K1  ; CART CONV STOP SNR On_State
1299  LD      SM400  ; Alway on bit
      ANI     X13C  ; CART CONV STOP SENSOR_S11
      MPS
      AND     T619  ; CART CONV STOP SNR Off_State
      RST     M618  ; CART CONV STOP SNR On_State
      MPP
      OUT     T619 K3  ; CART CONV STOP SNR Off_State
1309  LD      SM400  ; Alway on bit
      AND     Y150  ; VESSEL CONV FWD_INV6
      AND     X123  ; INVERTER6 RUN CHECK_VESSEL CONV
      MPS
      AND     T620  ; Vessel Conveyor FWD Run_State
      OUT     M620  ; Vessel Conveyor FWD Run_State
      MPP
      OUT     T620 K3  ; Vessel Conveyor FWD Run_State
1320  LD      SM400  ; Alway on bit
      AND     Y151  ; VESSEL CONV BWD_INV6
      AND     X123  ; INVERTER6 RUN CHECK_VESSEL CONV
      MPS
      AND     T621  ; Vessel Conveyor BWD Run_State
      OUT     M621  ; Vessel Conveyor BWD Run_State
      MPP
      OUT     T621 K3  ; Vessel Conveyor BWD Run_State
1331  LD      SM400  ; Alway on bit
      AND     Y158  ; CART CONV FWD_INV8
      AND     X125  ; INVERTER8 RUN CHECK_CART CONV
      MPS
      AND     T622  ; CART Conveyor FWD Run_State
      OUT     M622  ; CART Conveyor FWD Run_State
      MPP
      OUT     T622 K3  ; CART Conveyor FWD Run_State
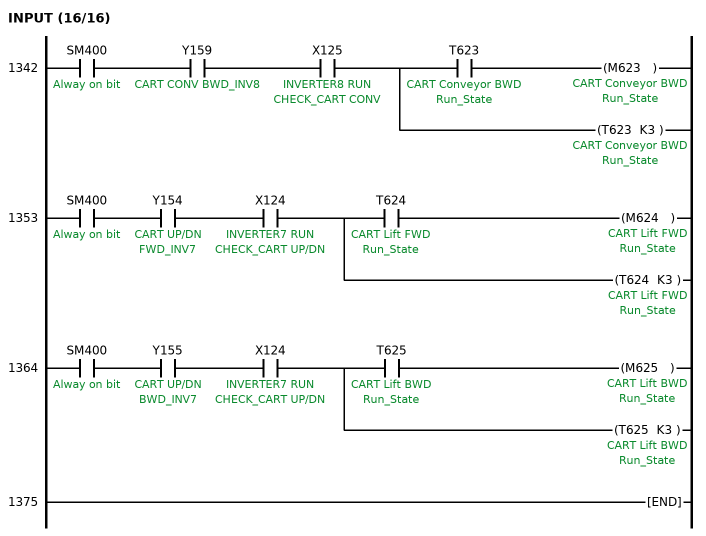
1342  LD      SM400  ; Alway on bit
      AND     Y159  ; CART CONV BWD_INV8
      AND     X125  ; INVERTER8 RUN CHECK_CART CONV
      MPS
      AND     T623  ; CART Conveyor BWD Run_State
      OUT     M623  ; CART Conveyor BWD Run_State
      MPP
      OUT     T623 K3  ; CART Conveyor BWD Run_State
1353  LD      SM400  ; Alway on bit
      AND     Y154  ; CART UP/DN FWD_INV7
      AND     X124  ; INVERTER7 RUN CHECK_CART UP/DN
      MPS
      AND     T624  ; CART Lift FWD Run_State
      OUT     M624  ; CART Lift FWD Run_State
      MPP
      OUT     T624 K3  ; CART Lift FWD Run_State
1364  LD      SM400  ; Alway on bit
      AND     Y155  ; CART UP/DN BWD_INV7
      AND     X124  ; INVERTER7 RUN CHECK_CART UP/DN
      MPS
      AND     T625  ; CART Lift BWD Run_State
      OUT     M625  ; CART Lift BWD Run_State
      MPP
      OUT     T625 K3  ; CART Lift BWD Run_State
1375  END
END_PROGRAM
